// TIA Portal V20 export
TYPE "zp_Tool_Data"
// stored: Namespace CITI_Logic
   STRUCT
      ToolPocketOrStaNumber : Int;   // Tool Pocket or Station Number
      SerialNumber : DInt;   // Serial Number
      ToolTypeOrGroup : String[12];   // Tool Type or Group
      MaximumToolLife : DInt;   // Maximum Tool Life
      ToolLifeWarningLimit : DInt;   // Tool Life Warning Limit
      ToolCyclesUsed : DInt;   // Tool Cycles Used
   END_STRUCT;
END_TYPE
